PROGRAM XTS
VAR
END_VAR

END_PROGRAM

(* stored: Version 1.1.0.1, ProductVersion 3.1.4024.12
   POU XTS: Id {74115216-9c4a-0cfc-0a38-bdb4d9dc9f35}, SpecialFunc None *)
